# EPICS substitutions: lensApp/Db/shutter.substitutions
file shutter.tpl-db
{
    {
        LOCATION = $(LOCATION)
        SHUTTER = $(SHUTTER)
    }
}
